// TIA Portal V20 export
TYPE "typeEm2Standard"
// stored: Access Published, Namespace Unit1
   STRUCT
      commands { ExternalWritable := 'False'} : "Unit1.typeEm2Commands";
      monitoring { ExternalWritable := 'False'} : "Unit1.typeEm2Monitoring";
   END_STRUCT;
END_TYPE
